FUNCTION_BLOCK FB_CheckHeartBeat
VAR_INPUT
	iHeartBeat		: UINT;
END_VAR
VAR_OUTPUT
	bOK				: BOOL;
END_VAR
VAR
	iHeartBeat_Old	: UINT;
	tofTimeOut		: TOF;
	tMaxTime		: TIME := T#500MS;
END_VAR


tofTimeOut(	IN := (iHeartBeat <> iHeartBeat_Old),
			PT := tMaxtime,
			Q => bOK);
iHeartBeat_Old := iHeartBeat;

PROPERTY PUBLIC P_tMaxTime : TIME
GET
P_tMaxTime := tMaxTime;
END_GET
SET
tMaxTime := P_tMaxTime;
END_SET
END_PROPERTY

END_FUNCTION_BLOCK

(* stored: Version 1.1.0.1, ProductVersion 3.1.4024.2
   POU FB_CheckHeartBeat: Id {aab34f87-4b56-4d23-8962-b2cf21baa8fd}, SpecialFunc None
   Property P_tMaxTime: Id {2cbed498-4cc6-4bf2-93bd-0f3018386df1}
   Get Get: Id {7ec62725-16bf-4bad-a850-82c04152be65}
   Set Set: Id {64990059-3e14-47a5-ad89-c3d3723db6f2} *)
